// TIA Portal project "LAB6.5" (V15)

(* hardware
DEVICE "S7-1200 station_1"  S7-1200 Station
   slot 0: "Rack_0"  S7-1200 Rack  Rack  V1.0
   slot 1: "PLC_1"  CPU 1214C DC/DC/DC  6ES7 214-1AG40-0XB0  V4.2
      slot 3: "AQ 1x12BIT_1"  AQ1 signal board  6ES7 232-4HA30-0XB0  V1.0
   slot 101: "CM 1243-5"  CM 1243-5  6GK7 243-5DX30-0XE0  V1.3
   slot 102: "CM 1241 (RS485)_1"  CM 1241 (RS485)  6ES7 241-1CH30-0XB0  V1.0
*)

// ===== PLC "PLC_1"  CPU 1214C DC/DC/DC =====

VAR_GLOBAL   // PLC tag table "Default tag table"
   "startZBOCZA" AT %I0.0 : Bool;
   "P_PRAG" AT %M10.0 : Bool;
   "resetZBOCZA" AT %I0.1 : Bool;
   "Tag_4" AT %M10.0 : Bool;
   "SPRZEZ" AT %M10.2 : Bool;
   "wy_GEN" AT %M10.3 : Bool;
   "RESET" AT %M10.5 : Bool;
   "wLICZNIKA" AT %MW20 : Int;
   "NASTAWA" AT %MD200 : Time;
END_VAR

// folder: System blocks/Program resources

DATA_BLOCK "T1"   // DB1
{ S7_Optimized_Access := 'TRUE' }
AUTHOR : Simatic
FAMILY : IEC
NAME : IEC_TMR
VERSION : 1.0
// stored: InstanceOfName IEC_TIMER
"IEC_TIMER"
BEGIN
END_DATA_BLOCK

DATA_BLOCK "T2"   // DB2
{ S7_Optimized_Access := 'TRUE' }
AUTHOR : Simatic
FAMILY : IEC
NAME : IEC_TMR
VERSION : 1.0
// stored: InstanceOfName IEC_TIMER
"IEC_TIMER"
BEGIN
END_DATA_BLOCK

DATA_BLOCK "LICZNIK1"   // DB3
{ S7_Optimized_Access := 'TRUE' }
AUTHOR : Simatic
FAMILY : IEC
NAME : CNTR
VERSION : 1.0
// stored: InstanceOfName IEC_COUNTER
"IEC_COUNTER"
BEGIN
END_DATA_BLOCK

// folder: (top level)

ORGANIZATION_BLOCK "Main"   // OB1, LAD, ProgramCycle
TITLE = "Main Program Sweep (Cycle)"
{ S7_Optimized_Access := 'TRUE' }
VERSION : 0.1
// zbuduj generator pracujacy na wyj q1.0 w nastepujacy sposob generuje 10 impulsow o f = 2Hz i 5 impulsow o f 0.5 Hz
   VAR_INPUT
      Initial_Call : Bool;   // Initial call of this OB
      Remanence : Bool;   // =True, if remanent data are available
   END_VAR
BEGIN

REGION Network 1
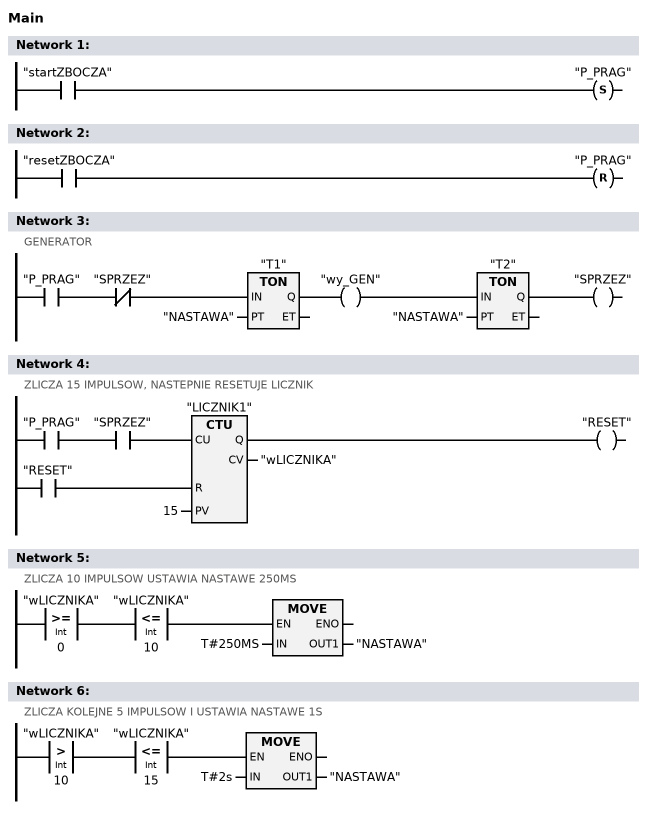
   RUNG wire#powerrail
      Contact( "startZBOCZA" )
      S_Coil( "P_PRAG" )
   END_RUNG
   // the same network as SCL:
   IF "startZBOCZA" THEN "P_PRAG" := TRUE; END_IF;
END_REGION

REGION Network 2
   RUNG wire#powerrail
      Contact( "resetZBOCZA" )
      R_Coil( "P_PRAG" )
   END_RUNG
   // the same network as SCL:
   IF "resetZBOCZA" THEN "P_PRAG" := FALSE; END_IF;
END_REGION

REGION Network 3
   // GENERATOR
   "T1".TON(IN := "P_PRAG" AND NOT "SPRZEZ", PT := "NASTAWA");
   "wy_GEN" := "T1".Q;
   "T2".TON(IN := "T1".Q, PT := "NASTAWA");
   "SPRZEZ" := "T2".Q;
END_REGION

REGION Network 4
   // ZLICZA 15 IMPULSOW, NASTEPNIE RESETUJE LICZNIK
   "LICZNIK1".CTU(CU := "P_PRAG" AND "SPRZEZ", R := "RESET", PV := 15, CV => "wLICZNIKA");
   "RESET" := "LICZNIK1".Q;
END_REGION

REGION Network 5
   // ZLICZA 10 IMPULSOW USTAWIA NASTAWE 250MS
   RUNG wire#powerrail
      { S7_Templates := "SrcType := Int" } GE_Contact(in1 := "wLICZNIKA", in2 := 0)
      { S7_Templates := "SrcType := Int" } LE_Contact(in1 := "wLICZNIKA", in2 := 10)
      Move(in := T#250MS, out1 => "NASTAWA")
   END_RUNG
   // the same network as SCL:
   IF ("wLICZNIKA" >= 0) AND ("wLICZNIKA" <= 10) THEN "NASTAWA" := T#250MS; END_IF;
END_REGION

REGION Network 6
   // ZLICZA KOLEJNE 5 IMPULSOW I USTAWIA NASTAWE 1S
   RUNG wire#powerrail
      { S7_Templates := "SrcType := Int" } GT_Contact(in1 := "wLICZNIKA", in2 := 10)
      { S7_Templates := "SrcType := Int" } LE_Contact(in1 := "wLICZNIKA", in2 := 15)
      Move(in := T#2s, out1 => "NASTAWA")
   END_RUNG
   // the same network as SCL:
   IF ("wLICZNIKA" > 10) AND ("wLICZNIKA" <= 15) THEN "NASTAWA" := T#2s; END_IF;
END_REGION
END_ORGANIZATION_BLOCK